FUNCTION_BLOCK FB_TestRound EXTENDS TcUnit.FB_TestSuite

//REAL
testRoundRealFail();
testRoundRealSuccess();
testRoundRealToHigh();

// LREAL
testRoundLREALFail();
testRoundLREALSuccess();
testRoundLREALToHigh();

METHOD testRoundLREALFail
VAR
	rValue 		: LREAL := 1000.222222;
	Actual		: LREAL;
	Expected  	: LREAL;
END_VAR
TEST('testRoundLREALFail');

// Act
Actual := 1000.222; 

// Arrange
Expected := 1000.22;

// Assert
AssertFalse( Condition := Expected = Actual, 
			 Message := 'testRoundLREALFail Failed to round LREAL');
			 
			 
			 
TEST_FINISHED();
END_METHOD

METHOD testRoundLREALSuccess
VAR
	rValue 		: LREAL := 1000.222222;
	Actual		: LREAL;
	Expected  	: LREAL;
END_VAR
TEST('testRoundLREALSuccess');

// Act
Actual := F_ROUNDLREAL(rValue, 2); 

// Arrange
Expected := 1000.22;

// Assert
AssertEquals(Expected := Expected, 
			 Actual := Actual,
			 Message := 'testRoundLREALSuccess Failed to round LREAL');
			 
			 
			 
TEST_FINISHED();
END_METHOD

METHOD testRoundLREALToHigh
VAR
	rValue 		: LREAL := 1000.226666;
	Actual		: LREAL;
	Expected  	: LREAL;
END_VAR
TEST('testRoundLREALToHigh');

// Act
Actual := F_ROUNDLREAL(rValue, 2); 

// Arrange
Expected := 1000.23;

// Assert
AssertEquals_LREAL( Expected :=  Expected, 
				Actual := Actual,
				Delta := 0.00,
			 	Message := 'testRoundLREALToHigh Failed to round LREAL');
			 
			 
			 
TEST_FINISHED();
END_METHOD

METHOD testRoundRealFail
VAR
	rValue 		: REAL := 1000.222222;
	Actual		: REAL;
	Expected  	: REAL;
END_VAR
TEST('testRoundRealFail');

// Act
Actual := 1000.222; 

// Arrange
Expected := 1000.22;

// Assert
AssertFalse( Condition := Expected = Actual, 
			 Message := 'testRoundRealFail Failed to round REAL');
			 
			 
			 
TEST_FINISHED();
END_METHOD

METHOD testRoundRealSuccess
VAR
	rValue 		: REAL := 1000.22222;
	Actual		: REAL;
	Expected  	: REAL;
END_VAR
TEST('testRoundRealSuccess');

// Act
Actual := F_ROUNDREAL(rValue, 2); 

// Arrange
Expected := 1000.22;

// Assert
AssertEquals(Expected := Expected, 
			 Actual := Actual,
			 Message := 'testRoundRealSuccess Failed to round REAL');
			 
			 
			 
TEST_FINISHED();
END_METHOD

METHOD testRoundRealToHigh
VAR
	rValue 		: REAL := 1000.226666;
	Actual		: REAL;
	Expected  	: REAL;
END_VAR
TEST('testRoundRealToHigh');

// Act
Actual := F_ROUNDREAL(rValue, 2); 

// Arrange
Expected := 1000.23;

// Assert
AssertEquals_REAL( Expected :=  Expected, 
				Actual := Actual,
				Delta := 0.00,
			 	Message := 'testRoundRealToHigh Failed to round REAL');
			 
			 
			 
TEST_FINISHED();
END_METHOD

END_FUNCTION_BLOCK

(* stored: Version 1.1.0.1, ProductVersion 3.1.4024.9
   POU FB_TestRound: Id {92000e0b-3a08-4346-91c0-8b471b1ff965}, SpecialFunc None
   Method testRoundLREALFail: Id {75a07223-c3fb-4fe9-9720-e7d1da3e7f14}
   Method testRoundLREALSuccess: Id {56bbe050-808e-4c28-80dd-438051f9d06c}
   Method testRoundLREALToHigh: Id {9448a483-1a90-427c-b183-181b75054701}
   Method testRoundRealFail: Id {ce530fdf-2fc4-48d5-a14b-9756c10cbeca}
   Method testRoundRealSuccess: Id {972e2527-061b-4f8b-979d-4770a9b664a6}
   Method testRoundRealToHigh: Id {18226e24-f317-455d-881a-ac6cfcd9211b} *)
